(* PLC project motor_test1, Beckhoff Automation GmbH TwinCAT PLC Control 3.5.6.0 *)
(* stored: creationDateTime 2015-12-12T13:32:27.246457, modificationDateTime 2015-12-12T13:32:27.2494689 *)

PROGRAM allgemein

                        (*safe the min and max value of the force*)
                            IF maxForceValuePos < acutalForceValue THEN
                            maxForceValuePos := acutalForceValue;
                            END_IF
                            IF maxForceValueNeg > acutalForceValue THEN
                            maxForceValueNeg := acutalForceValue;
                            END_IF
                    
END_PROGRAM
